# EPICS substitutions: db/Beckhoff_7XXX/ecmcEL7037_PosIF.substitutions
file "ecmcEL7037_PosIF-chX.template"
{
  pattern {CH_ID}
          {01   }
}
